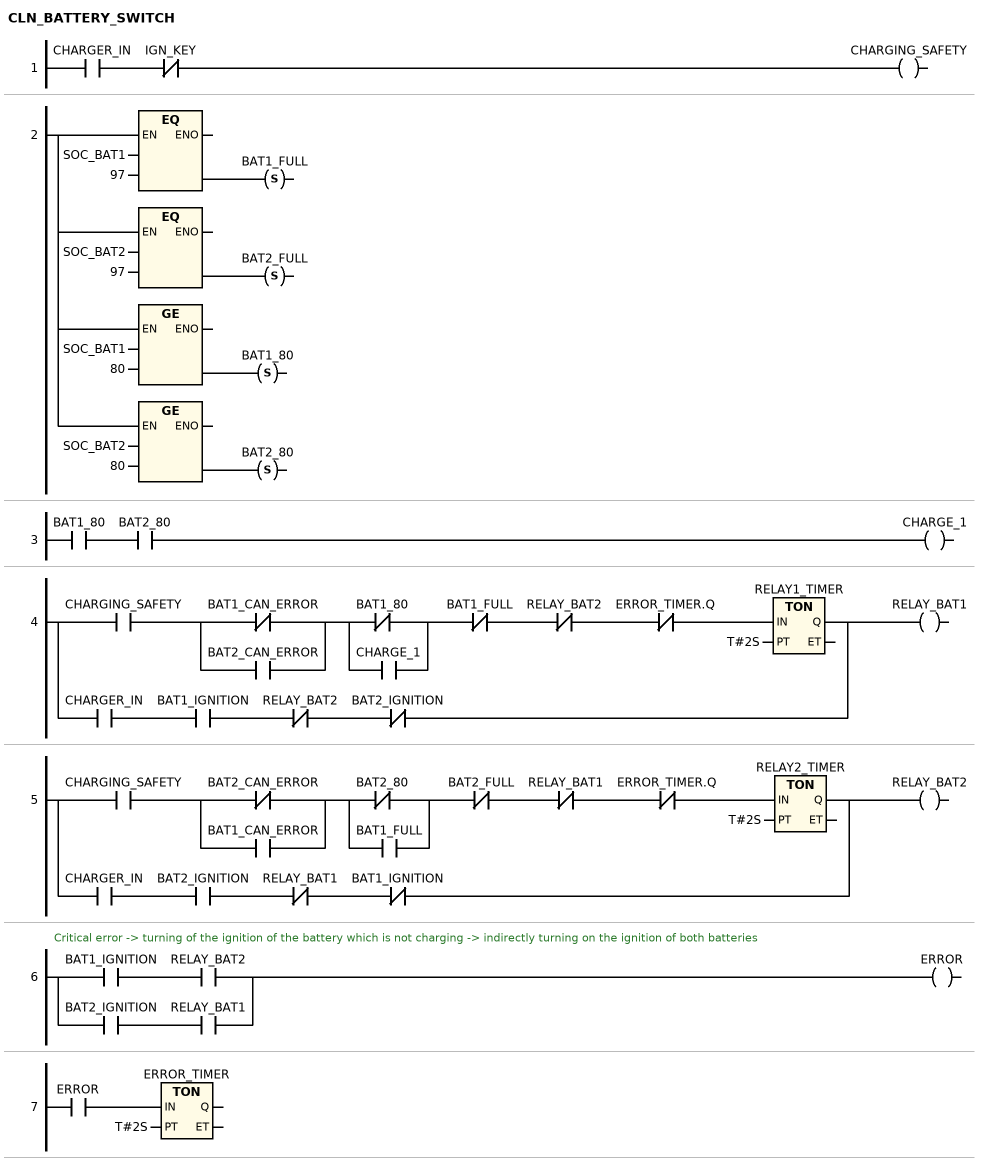
[picture p24: CLN_BATTERY_SWITCH (LD)]
_LD_ (* Ladder Diagram *)
NETWORK 1
	[CHARGER_IN] - [/IGN_KEY] --- (CHARGING_SAFETY)
NETWORK 2
	*
		EN --- EQ(SOC_BAT1, 97) => S BAT1_FULL
		EN --- EQ(SOC_BAT2, 97) => S BAT2_FULL
		EN --- GE(SOC_BAT1, 80) => S BAT1_80
		EN --- GE(SOC_BAT2, 80) => S BAT2_80
NETWORK 3
	[BAT1_80] - [BAT2_80] --- (CHARGE_1)
NETWORK 4
	{ [CHARGING_SAFETY] - { [/BAT1_CAN_ERROR] | [BAT2_CAN_ERROR] } - { [/BAT1_80] | [CHARGE_1] } - [/BAT1_FULL] - [/RELAY_BAT2] - [/ERROR_TIMER.Q] - RELAY1_TIMER:TON(IN: *, PT: T#2S) | [CHARGER_IN] - [BAT1_IGNITION] - [/RELAY_BAT2] - [/BAT2_IGNITION] } --- (RELAY_BAT1)
NETWORK 5
	{ [CHARGING_SAFETY] - { [/BAT2_CAN_ERROR] | [BAT1_CAN_ERROR] } - { [/BAT2_80] | [BAT1_FULL] } - [/BAT2_FULL] - [/RELAY_BAT1] - [/ERROR_TIMER.Q] - RELAY2_TIMER:TON(IN: *, PT: T#2S) | [CHARGER_IN] - [BAT2_IGNITION] - [/RELAY_BAT1] - [/BAT1_IGNITION] } --- (RELAY_BAT2)
NETWORK 6 (* Critical error -> turning of the ignition of the battery which is not charging -> indirectly turning on the ignition of both batteries *)
	{ [BAT1_IGNITION] - [RELAY_BAT2] | [BAT2_IGNITION] - [RELAY_BAT1] } --- (ERROR)
NETWORK 7
	[ERROR] - ERROR_TIMER:TON(IN: *, PT: T#2S)
_END_LD_
(* the same logic as Structured Text *)
(* Network 1 *)
CHARGING_SAFETY := CHARGER_IN AND NOT IGN_KEY;
(* Network 2 *)
IF SOC_BAT1 = 97 THEN BAT1_FULL := TRUE; END_IF;
IF SOC_BAT2 = 97 THEN BAT2_FULL := TRUE; END_IF;
IF SOC_BAT1 >= 80 THEN BAT1_80 := TRUE; END_IF;
IF SOC_BAT2 >= 80 THEN BAT2_80 := TRUE; END_IF;
(* Network 3 *)
CHARGE_1 := BAT1_80 AND BAT2_80;
(* Network 4 *)
RELAY1_TIMER(IN := CHARGING_SAFETY AND (NOT BAT1_CAN_ERROR OR BAT2_CAN_ERROR) AND (NOT BAT1_80 OR CHARGE_1) AND NOT BAT1_FULL AND NOT RELAY_BAT2 AND NOT ERROR_TIMER.Q, PT := T#2S);
RELAY_BAT1 := RELAY1_TIMER.Q OR CHARGER_IN AND BAT1_IGNITION AND NOT RELAY_BAT2 AND NOT BAT2_IGNITION;
(* Network 5 *)
RELAY2_TIMER(IN := CHARGING_SAFETY AND (NOT BAT2_CAN_ERROR OR BAT1_CAN_ERROR) AND (NOT BAT2_80 OR BAT1_FULL) AND NOT BAT2_FULL AND NOT RELAY_BAT1 AND NOT ERROR_TIMER.Q, PT := T#2S);
RELAY_BAT2 := RELAY2_TIMER.Q OR CHARGER_IN AND BAT2_IGNITION AND NOT RELAY_BAT1 AND NOT BAT1_IGNITION;
(* Network 6: Critical error -> turning of the ignition of the battery which is not charging -> indirectly turning on the ignition of both batteries *)
ERROR := BAT1_IGNITION AND RELAY_BAT2 OR BAT2_IGNITION AND RELAY_BAT1;
(* Network 7 *)
ERROR_TIMER(IN := ERROR, PT := T#2S);
END_FUNCTION_BLOCK

(* POU PROGRAM_FBs/CLN_CHARGING, LD *)
FUNCTION_BLOCK CLN_CHARGING
(*
THIS BLOCK IS COMPATIBLE FOR 2X CLN BATTERIES0

Created BY: Adiga
Date: 25-01-24
UPDATED :14-03-25
Version: 4
1.DUAL BATTERY CAHRGING BLOCK ONLY FOR CLN
2.UPDATED THE BLOCK FOR CHARGING WITH AND WITHOUT IGN ON
3.ADDED BATTERY CAN ERROR CODITION TO CHARGE
4.ADDED TIMER BEFORE SWITCHING BATTRY BELAY.
.
*)

VAR_INPUT
	CHANNEL: BYTE;
	CHARGER_IN: BOOL;
	IGN_KEY: BOOL;
	BAT1_IGN: BOOL;
	BAT2_IGN: BOOL;
	SOC1: BYTE;
	SOC2: BYTE;
	BAT_CAN_ERROR1: BOOL;
	BAT_CAN_ERROR2: BOOL;
	BATTERY_CHARGING: BOOL;
END_VAR

VAR_OUTPUT
	RELAY_BAT1: BOOL;
	RELAY_BAT2: BOOL;
	BLUE_LED_OUT: BOOL;
	ERROR: BOOL;
	BUZZER_ON: BOOL;
	CHARGING1: BOOL;
	CHARGING2: BOOL;
END_VAR

VAR
	CHARGE_1: BOOL;
	BAT_1_FULL: BOOL;
	BAT_2_FULL: BOOL;
	T1: TON;
	T2: TON;
	T3: TON;
	IGNITION_OFF: BOOL;
	BAT_1_80: BOOL;
	BAT_2_80: BOOL;
	FTRIG1: F_TRIG;
	TIMER5: TON;
	T4: TON;
	T5: TON;
	CHARGING_2: BLINK;
	CHARGING_1: BLINK;
END_VAR
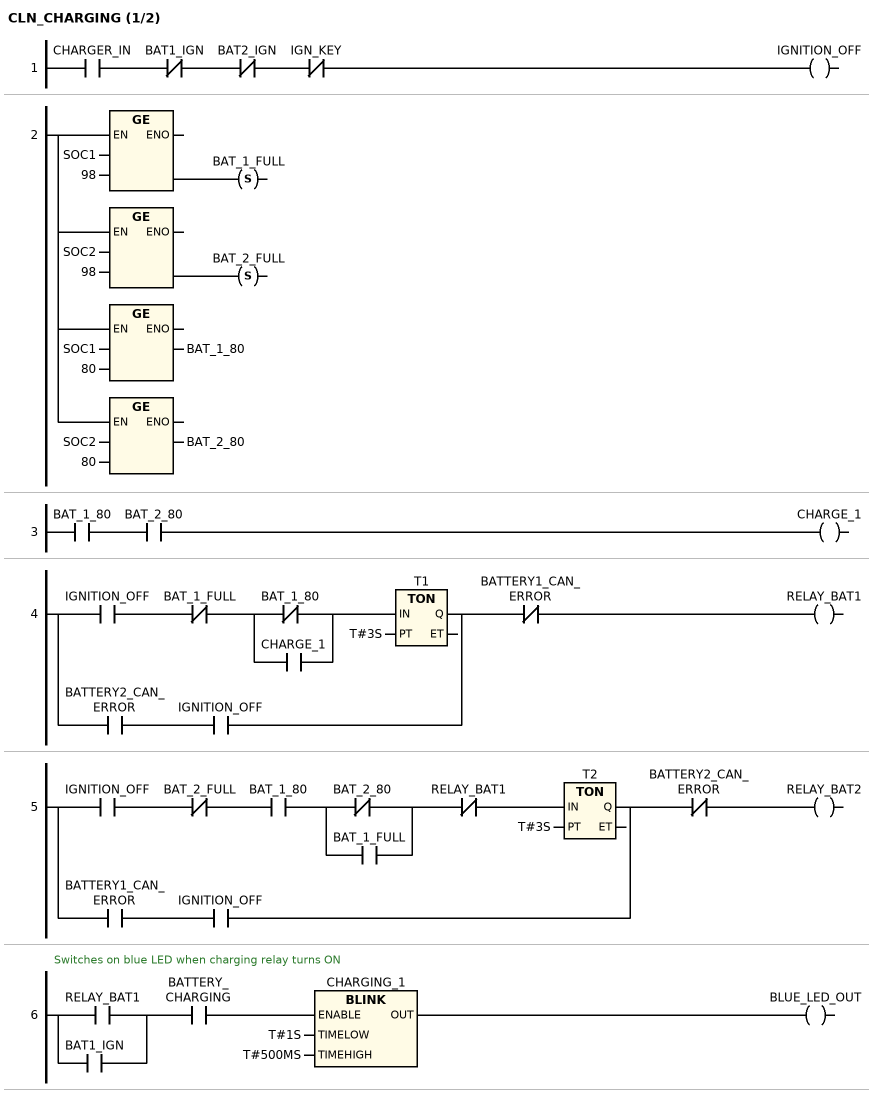
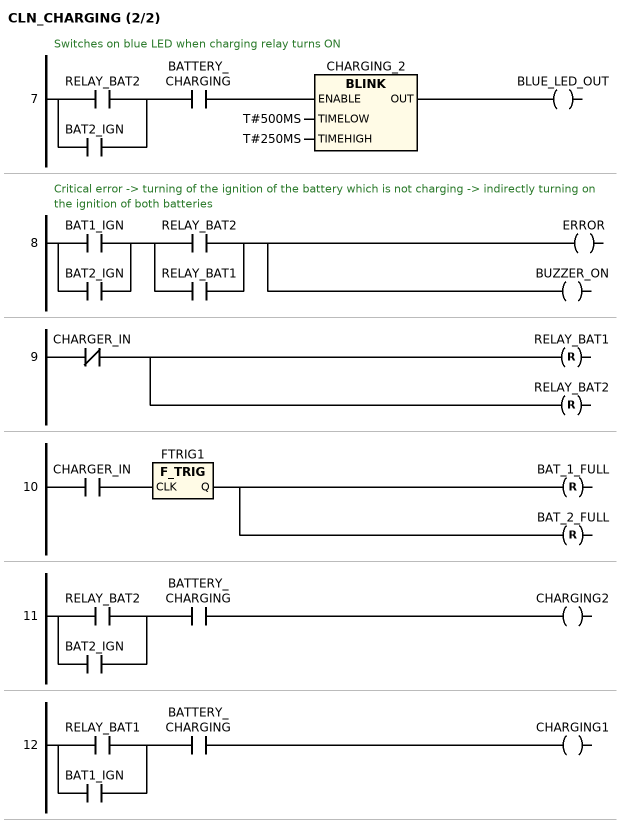
_LD_ (* Ladder Diagram *)
NETWORK 1
	[CHARGER_IN] - [/BAT1_IGN] - [/BAT2_IGN] - [/IGN_KEY] --- (IGNITION_OFF)
NETWORK 2
	*
		EN --- GE(SOC1, 98) => S BAT_1_FULL
		EN --- GE(SOC2, 98) => S BAT_2_FULL
		EN --- GE(SOC1, 80) => BAT_1_80
		EN --- GE(SOC2, 80) => BAT_2_80
NETWORK 3
	[BAT_1_80] - [BAT_2_80] --- (CHARGE_1)
NETWORK 4
	{ [IGNITION_OFF] - [/BAT_1_FULL] - { [/BAT_1_80] | [CHARGE_1] } - T1:TON(IN: *, PT: T#3S) | [BATTERY2_CAN_ERROR] - [IGNITION_OFF] } - [/BATTERY1_CAN_ERROR] --- (RELAY_BAT1)
NETWORK 5
	{ [IGNITION_OFF] - [/BAT_2_FULL] - [BAT_1_80] - { [/BAT_2_80] | [BAT_1_FULL] } - [/RELAY_BAT1] - T2:TON(IN: *, PT: T#3S) | [BATTERY1_CAN_ERROR] - [IGNITION_OFF] } - [/BATTERY2_CAN_ERROR] --- (RELAY_BAT2)
NETWORK 6 (* Switches on blue LED when charging relay turns ON *)
	{ [RELAY_BAT1] | [BAT1_IGN] } - [BATTERY_CHARGING] - CHARGING_1:BLINK(ENABLE: *, TIMELOW: T#1S, TIMEHIGH: T#500MS) --- (BLUE_LED_OUT)
NETWORK 7 (* Switches on blue LED when charging relay turns ON *)
	{ [RELAY_BAT2] | [BAT2_IGN] } - [BATTERY_CHARGING] - CHARGING_2:BLINK(ENABLE: *, TIMELOW: T#500MS, TIMEHIGH: T#250MS) --- (BLUE_LED_OUT)
NETWORK 8 (* Critical error -> turning of the ignition of the battery which is not charging -> indirectly turning on the ignition of both batteries *)
	{ [BAT1_IGN] | [BAT2_IGN] } - { [RELAY_BAT2] | [RELAY_BAT1] } --- (ERROR) (BUZZER_ON)
NETWORK 9
	[/CHARGER_IN] --- (R RELAY_BAT1) (R RELAY_BAT2)
NETWORK 10
	[CHARGER_IN] - FTRIG1:F_TRIG(CLK: *) --- (R BAT_1_FULL) (R BAT_2_FULL)
NETWORK 11
	{ [RELAY_BAT2] | [BAT2_IGN] } - [BATTERY_CHARGING] --- (CHARGING2)
NETWORK 12
	{ [RELAY_BAT1] | [BAT1_IGN] } - [BATTERY_CHARGING] --- (CHARGING1)
_END_LD_
(* the same logic as Structured Text *)
(* Network 1 *)
IGNITION_OFF := CHARGER_IN AND NOT BAT1_IGN AND NOT BAT2_IGN AND NOT IGN_KEY;
(* Network 2 *)
IF SOC1 >= 98 THEN BAT_1_FULL := TRUE; END_IF;
IF SOC2 >= 98 THEN BAT_2_FULL := TRUE; END_IF;
BAT_1_80 := SOC1 >= 80;
BAT_2_80 := SOC2 >= 80;
(* Network 3 *)
CHARGE_1 := BAT_1_80 AND BAT_2_80;
(* Network 4 *)
T1(IN := IGNITION_OFF AND NOT BAT_1_FULL AND (NOT BAT_1_80 OR CHARGE_1), PT := T#3S);
RELAY_BAT1 := (T1.Q OR BATTERY2_CAN_ERROR AND IGNITION_OFF) AND NOT BATTERY1_CAN_ERROR;
(* Network 5 *)
T2(IN := IGNITION_OFF AND NOT BAT_2_FULL AND BAT_1_80 AND (NOT BAT_2_80 OR BAT_1_FULL) AND NOT RELAY_BAT1, PT := T#3S);
RELAY_BAT2 := (T2.Q OR BATTERY1_CAN_ERROR AND IGNITION_OFF) AND NOT BATTERY2_CAN_ERROR;
(* Network 6: Switches on blue LED when charging relay turns ON *)
CHARGING_1(ENABLE := (RELAY_BAT1 OR BAT1_IGN) AND BATTERY_CHARGING, TIMELOW := T#1S, TIMEHIGH := T#500MS);
BLUE_LED_OUT := CHARGING_1.OUT;
(* Network 7: Switches on blue LED when charging relay turns ON *)
CHARGING_2(ENABLE := (RELAY_BAT2 OR BAT2_IGN) AND BATTERY_CHARGING, TIMELOW := T#500MS, TIMEHIGH := T#250MS);
BLUE_LED_OUT := CHARGING_2.OUT;
(* Network 8: Critical error -> turning of the ignition of the battery which is not charging -> indirectly turning on the ignition of both batteries *)
ERROR := (BAT1_IGN OR BAT2_IGN) AND (RELAY_BAT2 OR RELAY_BAT1);
BUZZER_ON := ERROR;
(* Network 9 *)
IF NOT CHARGER_IN THEN RELAY_BAT1 := FALSE; RELAY_BAT2 := FALSE; END_IF;
(* Network 10 *)
FTRIG1(CLK := CHARGER_IN);
IF FTRIG1.Q THEN BAT_1_FULL := FALSE; BAT_2_FULL := FALSE; END_IF;
(* Network 11 *)
CHARGING2 := (RELAY_BAT2 OR BAT2_IGN) AND BATTERY_CHARGING;
(* Network 12 *)
CHARGING1 := (RELAY_BAT1 OR BAT1_IGN) AND BATTERY_CHARGING;
END_FUNCTION_BLOCK

(* POU PROGRAM_FBs/DRIVE_LOGIC, LD *)
FUNCTION_BLOCK DRIVE_LOGIC
VAR_INPUT
	JX: INT;
	JY: INT;
	LEFT_BUTTON: BOOL;
	JOY_ORIGIN: BOOL;
	EM_SWITCH_IN: BOOL;
	OVER_TEMP: BOOL;
END_VAR
VAR_OUTPUT
	JX_1: INT;
	JY_1: INT;
	DISARM: BOOL;
	EM_BRAKE_OUT: BOOL;
	DRIVE_ERROR: BOOL;
END_VAR
VAR
	SLEEP_TIMER: TON;
	ON_DELAY: TON;
	APPLY_EM: BOOL;
	LOW_RPM: BOOL;
	EMFB_ERROR: BOOL;
END_VAR
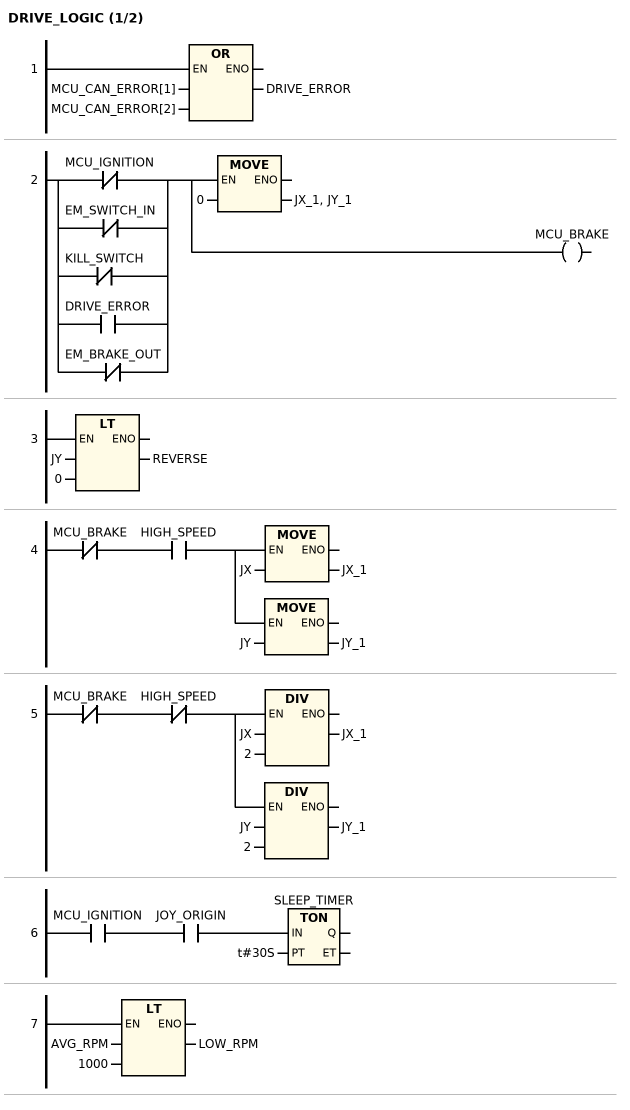
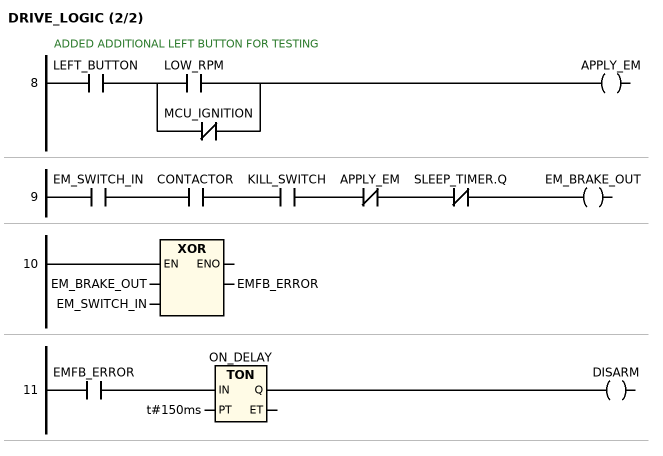
_LD_ (* Ladder Diagram *)
NETWORK 1
	*
		EN --- OR(MCU_CAN_ERROR[1], MCU_CAN_ERROR[2]) => DRIVE_ERROR
NETWORK 2
	{ [/MCU_IGNITION] | [/EM_SWITCH_IN] | [/KILL_SWITCH] | [DRIVE_ERROR] | [/EM_BRAKE_OUT] } --- (MCU_BRAKE)
		EN --- MOVE(0) => JX_1, JY_1
NETWORK 3
	*
		EN --- LT(JY, 0) => REVERSE
NETWORK 4
	[/MCU_BRAKE] - [HIGH_SPEED]
		EN --- MOVE(JX) => JX_1
		EN --- MOVE(JY) => JY_1
NETWORK 5
	[/MCU_BRAKE] - [/HIGH_SPEED]
		EN --- DIV(JX, 2) => JX_1
		EN --- DIV(JY, 2) => JY_1
NETWORK 6
	[MCU_IGNITION] - [JOY_ORIGIN] - SLEEP_TIMER:TON(IN: *, PT: t#30S)
NETWORK 7
	*
		EN --- LT(AVG_RPM, 1000) => LOW_RPM
NETWORK 8 (* ADDED ADDITIONAL LEFT BUTTON FOR TESTING *)
	[LEFT_BUTTON] - { [LOW_RPM] | [/MCU_IGNITION] } --- (APPLY_EM)
NETWORK 9
	[EM_SWITCH_IN] - [CONTACTOR] - [KILL_SWITCH] - [/APPLY_EM] - [/SLEEP_TIMER.Q] --- (EM_BRAKE_OUT)
NETWORK 10
	*
		EN --- XOR(EM_BRAKE_OUT, EM_SWITCH_IN) => EMFB_ERROR
NETWORK 11
	[EMFB_ERROR] - ON_DELAY:TON(IN: *, PT: t#150ms) --- (DISARM)
_END_LD_
(* the same logic as Structured Text *)
(* Network 1 *)
DRIVE_ERROR := MCU_CAN_ERROR[1] OR MCU_CAN_ERROR[2];
(* Network 2: see the listing above *)
(* Network 3 *)
REVERSE := JY < 0;
(* Network 4 *)
IF NOT MCU_BRAKE AND HIGH_SPEED THEN
	JX_1 := JX;
	JY_1 := JY;
END_IF;
(* Network 5 *)
IF NOT MCU_BRAKE AND NOT HIGH_SPEED THEN
	JX_1 := JX / 2;
	JY_1 := JY / 2;
END_IF;
(* Network 6 *)
SLEEP_TIMER(IN := MCU_IGNITION AND JOY_ORIGIN, PT := t#30S);
(* Network 7 *)
LOW_RPM := AVG_RPM < 1000;
(* Network 8 *)
APPLY_EM := LEFT_BUTTON AND (LOW_RPM OR NOT MCU_IGNITION);
(* Network 9 *)
EM_BRAKE_OUT := EM_SWITCH_IN AND CONTACTOR AND KILL_SWITCH AND NOT APPLY_EM AND NOT SLEEP_TIMER.Q;
(* Network 10 *)
EMFB_ERROR := EM_BRAKE_OUT XOR EM_SWITCH_IN;
(* Network 11 *)
ON_DELAY(IN := EMFB_ERROR, PT := t#150ms);
DISARM := ON_DELAY.Q;
END_FUNCTION_BLOCK

(* POU PROGRAM_FBs/DUAL_CLN_CHARGING, LD *)
FUNCTION_BLOCK DUAL_CLN_CHARGING
(*
THIS BLOCK IS COMPATIBLE FOR 2X CLN BATTERIES

Created BY: Adiga
Date: 8-08-24
Version: 1
 
*)

VAR_INPUT
	CHANNEL: BYTE;
	CHARGER_IN: BOOL;
	BAT_CAN_ERROR1: BOOL;
	BAT_CAN_ERROR2: BOOL;
	BAT1_IGN: BOOL;
	BAT2_IGN: BOOL;
	BATTERY_CHARGING: BOOL;

END_VAR

VAR_OUTPUT
	RELAY_BAT1: BOOL;
	RELAY_BAT2: BOOL;
	BLUE_LED_OUT: BOOL;
	ERROR: BOOL;
	BUZZER_ON: BOOL;
	CHARGING1: BOOL;
	CHARGING2: BOOL;
END_VAR

VAR
	CHARGE_1: BOOL;
	BAT_1_FULL: BOOL;
	BAT_2_FULL: BOOL;
	RX_SOLTERRA: RX_CAN;
	CHARGER_TIMER: TON;
	SOLTERRA_TX: CAN_TX;
	CHARGING_FRAME: ARRAY [0..7] OF BYTE  := 16#03,16#25,16#01,16#5E,0,0,0,0;

	T1: TON;
	T2: TON;
	T3: TON;
	SOC2: BYTE;
	SOC1: BYTE;
	TX_CLN: CAN_TX;
	IGNITION_OFF: BOOL;
	BAT_1_80: BOOL;
	BAT_2_80: BOOL;
	FTRIG1: F_TRIG;
	TIMER5: TON;
	T4: TON;
	T5: TON;

	CHARGE: F_TRIG;
END_VAR
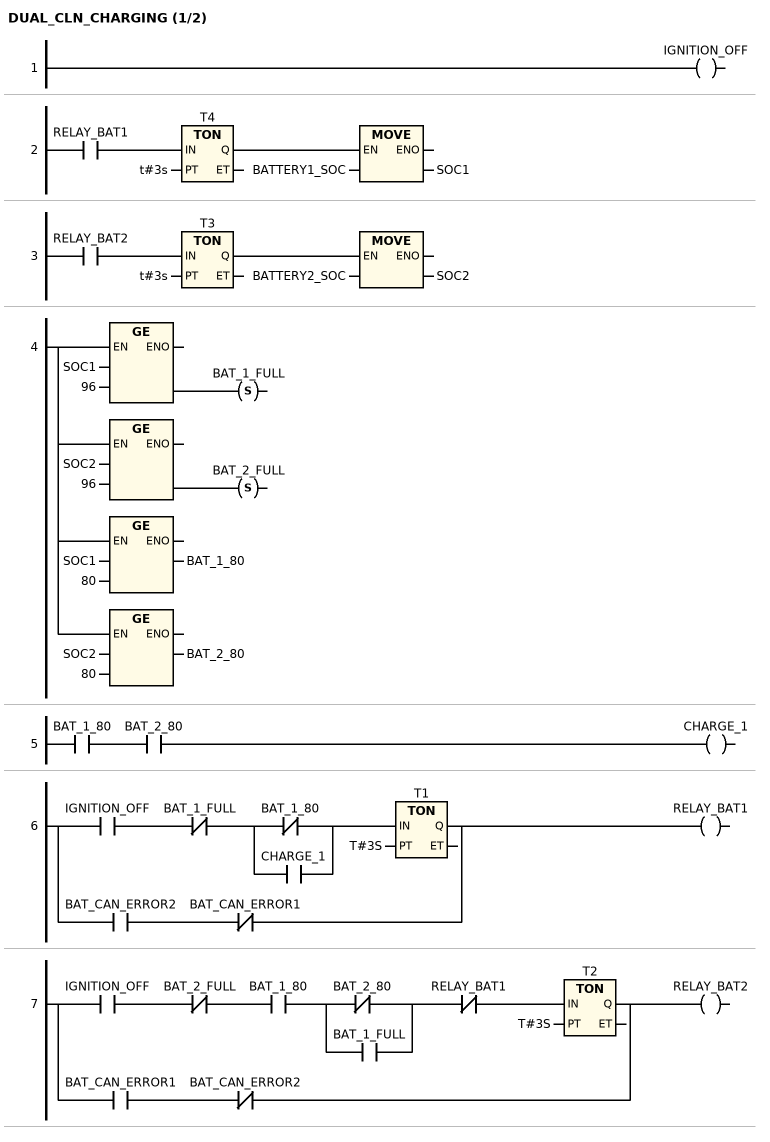
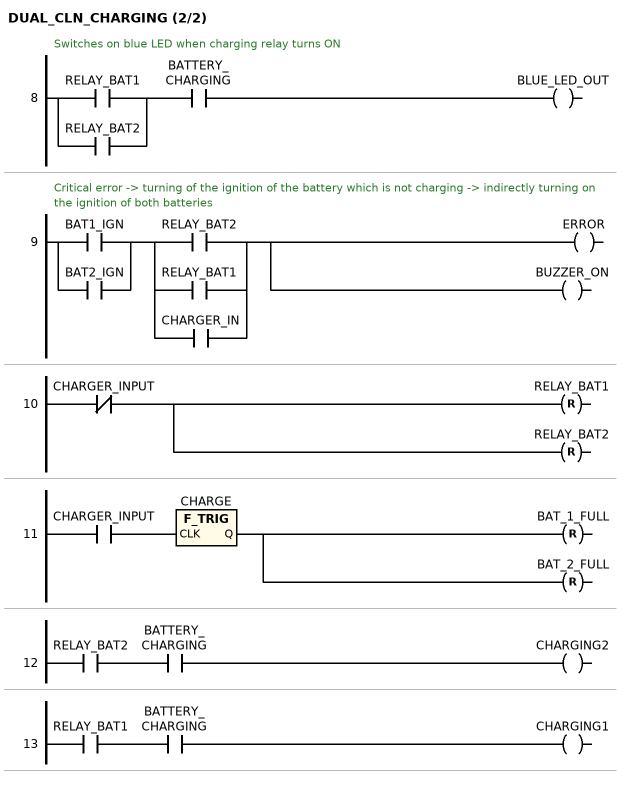
_LD_ (* Ladder Diagram *)
NETWORK 1
	* --- (IGNITION_OFF)
NETWORK 2
	[RELAY_BAT1] - T4:TON(IN: *, PT: t#3s)
		EN --- MOVE(BATTERY1_SOC) => SOC1
NETWORK 3
	[RELAY_BAT2] - T3:TON(IN: *, PT: t#3s)
		EN --- MOVE(BATTERY2_SOC) => SOC2
NETWORK 4
	*
		EN --- GE(SOC1, 96) => S BAT_1_FULL
		EN --- GE(SOC2, 96) => S BAT_2_FULL
		EN --- GE(SOC1, 80) => BAT_1_80
		EN --- GE(SOC2, 80) => BAT_2_80
NETWORK 5
	[BAT_1_80] - [BAT_2_80] --- (CHARGE_1)
NETWORK 6
	{ [IGNITION_OFF] - [/BAT_1_FULL] - { [/BAT_1_80] | [CHARGE_1] } - T1:TON(IN: *, PT: T#3S) | [BAT_CAN_ERROR2] - [/BAT_CAN_ERROR1] } --- (RELAY_BAT1)
NETWORK 7
	{ [IGNITION_OFF] - [/BAT_2_FULL] - [BAT_1_80] - { [/BAT_2_80] | [BAT_1_FULL] } - [/RELAY_BAT1] - T2:TON(IN: *, PT: T#3S) | [BAT_CAN_ERROR1] - [/BAT_CAN_ERROR2] } --- (RELAY_BAT2)
NETWORK 8 (* Switches on blue LED when charging relay turns ON *)
	{ [RELAY_BAT1] | [RELAY_BAT2] } - [BATTERY_CHARGING] --- (BLUE_LED_OUT)
NETWORK 9 (* Critical error -> turning of the ignition of the battery which is not charging -> indirectly turning on the ignition of both batteries *)
	{ [BAT1_IGN] | [BAT2_IGN] } - { [RELAY_BAT2] | [RELAY_BAT1] | [CHARGER_IN] } --- (ERROR) (BUZZER_ON)
NETWORK 10
	[/CHARGER_INPUT] --- (R RELAY_BAT1) (R RELAY_BAT2)
NETWORK 11
	[CHARGER_INPUT] - CHARGE:F_TRIG(CLK: *) --- (R BAT_1_FULL) (R BAT_2_FULL)
NETWORK 12
	[RELAY_BAT2] - [BATTERY_CHARGING] --- (CHARGING2)
NETWORK 13
	[RELAY_BAT1] - [BATTERY_CHARGING] --- (CHARGING1)
_END_LD_
(* the same logic as Structured Text *)
(* Network 1 *)
IGNITION_OFF := TRUE;
(* Network 2 *)
T4(IN := RELAY_BAT1, PT := t#3s);
IF T4.Q THEN
	SOC1 := BATTERY1_SOC;
END_IF;
(* Network 3 *)
T3(IN := RELAY_BAT2, PT := t#3s);
IF T3.Q THEN
	SOC2 := BATTERY2_SOC;
END_IF;
(* Network 4 *)
IF SOC1 >= 96 THEN BAT_1_FULL := TRUE; END_IF;
IF SOC2 >= 96 THEN BAT_2_FULL := TRUE; END_IF;
BAT_1_80 := SOC1 >= 80;
BAT_2_80 := SOC2 >= 80;
(* Network 5 *)
CHARGE_1 := BAT_1_80 AND BAT_2_80;
(* Network 6 *)
T1(IN := IGNITION_OFF AND NOT BAT_1_FULL AND (NOT BAT_1_80 OR CHARGE_1), PT := T#3S);
RELAY_BAT1 := T1.Q OR BAT_CAN_ERROR2 AND NOT BAT_CAN_ERROR1;
(* Network 7 *)
T2(IN := IGNITION_OFF AND NOT BAT_2_FULL AND BAT_1_80 AND (NOT BAT_2_80 OR BAT_1_FULL) AND NOT RELAY_BAT1, PT := T#3S);
RELAY_BAT2 := T2.Q OR BAT_CAN_ERROR1 AND NOT BAT_CAN_ERROR2;
(* Network 8: Switches on blue LED when charging relay turns ON *)
BLUE_LED_OUT := (RELAY_BAT1 OR RELAY_BAT2) AND BATTERY_CHARGING;
(* Network 9: Critical error -> turning of the ignition of the battery which is not charging -> indirectly turning on the ignition of both batteries *)
ERROR := (BAT1_IGN OR BAT2_IGN) AND (RELAY_BAT2 OR RELAY_BAT1 OR CHARGER_IN);
BUZZER_ON := ERROR;
(* Network 10 *)
IF NOT CHARGER_INPUT THEN RELAY_BAT1 := FALSE; RELAY_BAT2 := FALSE; END_IF;
(* Network 11 *)
CHARGE(CLK := CHARGER_INPUT);
IF CHARGE.Q THEN BAT_1_FULL := FALSE; BAT_2_FULL := FALSE; END_IF;
(* Network 12 *)
CHARGING2 := RELAY_BAT2 AND BATTERY_CHARGING;
(* Network 13 *)
CHARGING1 := RELAY_BAT1 AND BATTERY_CHARGING;
END_FUNCTION_BLOCK

(* POU FB_LIBRARY/DWORD_BYTE_CONVERSION, FBD *)
FUNCTION_BLOCK DWORD_BYTE_CONVERSION
(* BYTE_0 : LSB    ---------   BYTE_3 : MSB *)
VAR_INPUT
	INPUT_DWORD: DWORD;
END_VAR
VAR_OUTPUT
	BYTE_0: BYTE;
	BYTE_1: BYTE;
	BYTE_2: BYTE;
	BYTE_3: BYTE;
END_VAR
VAR
	WORD_1: WORD;
	WORD_2: WORD;
END_VAR
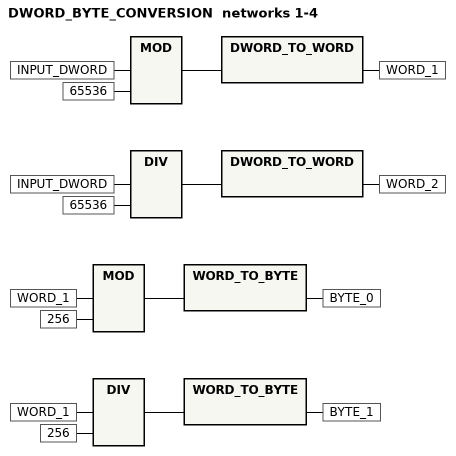
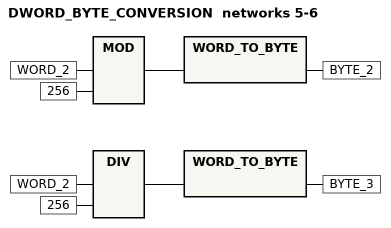
_FBD_ (* Function Block Diagram *)
NETWORK 1
	DWORD_TO_WORD(MOD(INPUT_DWORD, 65536)) => WORD_1
NETWORK 2
	DWORD_TO_WORD(DIV(INPUT_DWORD, 65536)) => WORD_2
NETWORK 3
	WORD_TO_BYTE(MOD(WORD_1, 256)) => BYTE_0
NETWORK 4
	WORD_TO_BYTE(DIV(WORD_1, 256)) => BYTE_1
NETWORK 5
	WORD_TO_BYTE(MOD(WORD_2, 256)) => BYTE_2
NETWORK 6
	WORD_TO_BYTE(DIV(WORD_2, 256)) => BYTE_3
_END_FBD_
(* the same logic as Structured Text *)
(* Network 1 *)
WORD_1 := DWORD_TO_WORD(INPUT_DWORD MOD 65536);
(* Network 2 *)
WORD_2 := DWORD_TO_WORD(INPUT_DWORD / 65536);
(* Network 3 *)
BYTE_0 := WORD_TO_BYTE(WORD_1 MOD 256);
(* Network 4 *)
BYTE_1 := WORD_TO_BYTE(WORD_1 / 256);
(* Network 5 *)
BYTE_2 := WORD_TO_BYTE(WORD_2 MOD 256);
(* Network 6 *)
BYTE_3 := WORD_TO_BYTE(WORD_2 / 256);
END_FUNCTION_BLOCK

(* POU PROGRAM_FBs/HYDRAULIC_CONTROL, LD *)
FUNCTION_BLOCK HYDRAULIC_CONTROL
VAR_INPUT
	DEADMAN: BOOL;
END_VAR
VAR_OUTPUT
END_VAR
VAR
	HYD_SPEED: INT;
	IDLE_MODE: BOOL;
	CUTOFF: INT;
	STATISTICS: STATISTICS_INT;
	RESET_AVG: BOOL;
	T1: TON;
	TRIG_1: R_TRIG;
	T2: TON;
	RUNNING_AVG: INT:=0;
	SET_IDLE: BOOL;
	HIGH_RPM: BOOL;
	WAIT: BOOL;
	UPPER_LIMIT: INT;
	MCU_RX_6: CHARA_MCU_RX;
	MCU_TX_6: CHARA_MCU_TX;
END_VAR
VAR CONSTANT
	IDLE_SPEED: INT :=0;
	ECO_CUTOFF: INT := 70;
	POWER_CUTOFF: INT := 90;
	BUFFER: INT := 10;
	HYD_RAMP: INT:= 100;
	MCU_RAMP: BYTE := 5;
	PHASE_LIMIT: BYTE := 60;
END_VAR
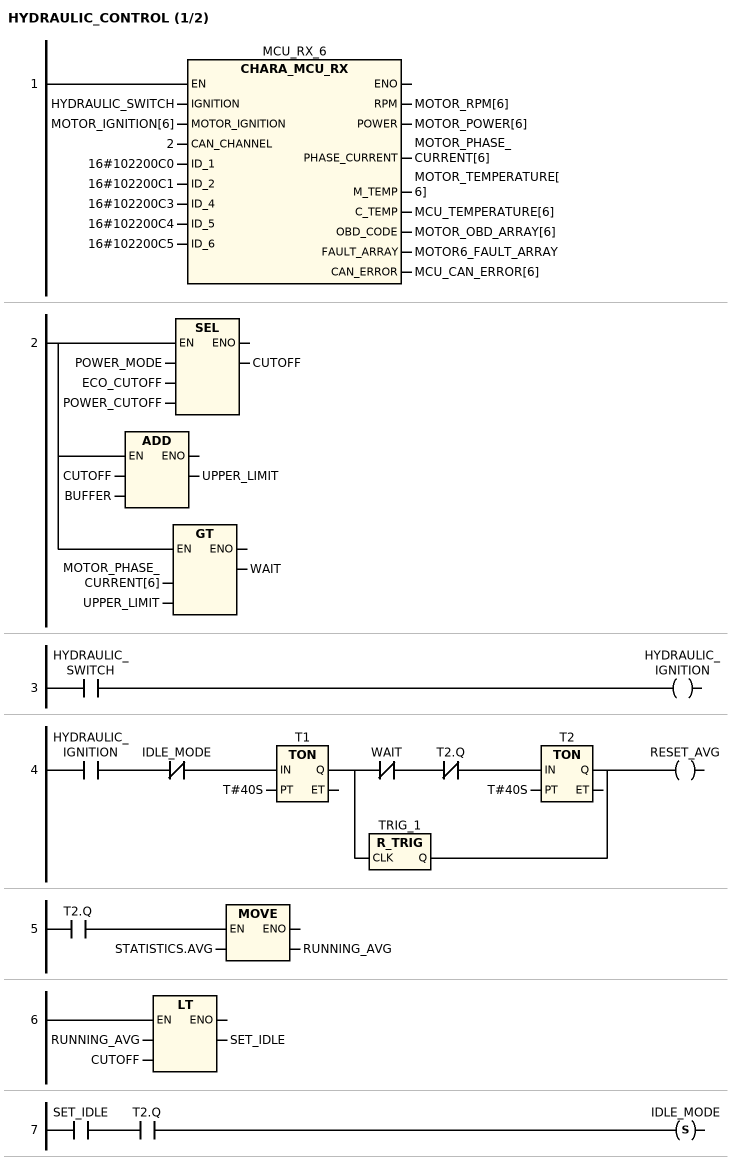
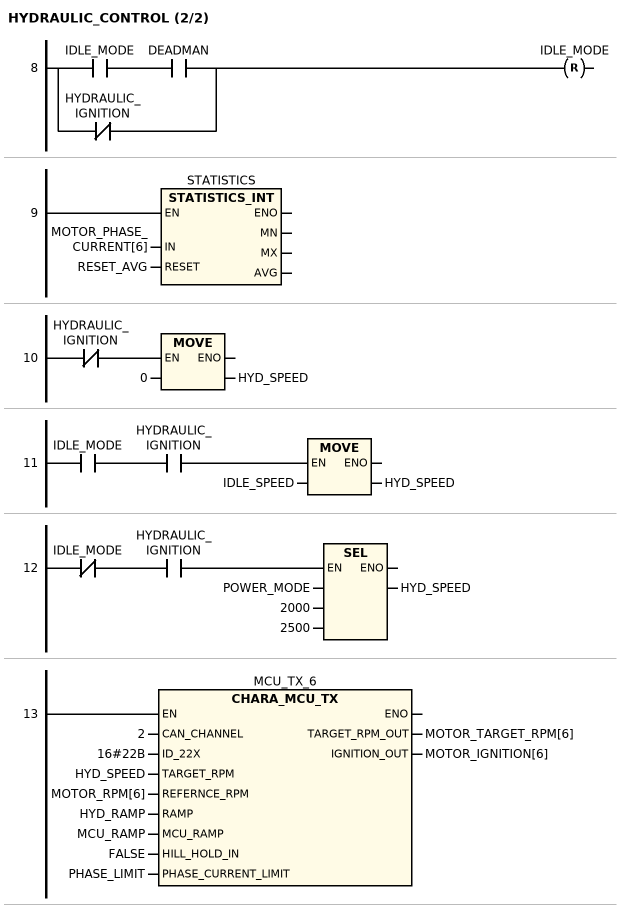
_LD_ (* Ladder Diagram *)
NETWORK 1
	*
		EN --- MCU_RX_6:CHARA_MCU_RX(IGNITION: HYDRAULIC_SWITCH, MOTOR_IGNITION: MOTOR_IGNITION[6], CAN_CHANNEL: 2, ID_1: 16#102200C0, ID_2: 16#102200C1, ID_4: 16#102200C3, ID_5: 16#102200C4, ID_6: 16#102200C5, POWER => MOTOR_POWER[6], PHASE_CURRENT => MOTOR_PHASE_CURRENT[6], M_TEMP => MOTOR_TEMPERATURE[6], C_TEMP => MCU_TEMPERATURE[6], OBD_CODE => MOTOR_OBD_ARRAY[6], FAULT_ARRAY => MOTOR6_FAULT_ARRAY, CAN_ERROR => MCU_CAN_ERROR[6]) => MOTOR_RPM[6]
NETWORK 2
	*
		EN --- SEL(POWER_MODE, ECO_CUTOFF, POWER_CUTOFF) => CUTOFF
		EN --- ADD(CUTOFF, BUFFER) => UPPER_LIMIT
		EN --- GT(MOTOR_PHASE_CURRENT[6], UPPER_LIMIT) => WAIT
NETWORK 3
	[HYDRAULIC_SWITCH] --- (HYDRAULIC_IGNITION)
NETWORK 4
	[HYDRAULIC_IGNITION] - [/IDLE_MODE] - T1:TON(IN: *, PT: T#40S) - { [/WAIT] - [/T2.Q] - T2:TON(IN: *, PT: T#40S) | TRIG_1:R_TRIG(CLK: *) } --- (RESET_AVG)
NETWORK 5
	[T2.Q]
		EN --- MOVE(STATISTICS.AVG) => RUNNING_AVG
NETWORK 6
	*
		EN --- LT(RUNNING_AVG, CUTOFF) => SET_IDLE
NETWORK 7
	[SET_IDLE] - [T2.Q] --- (S IDLE_MODE)
NETWORK 8
	{ [IDLE_MODE] - [DEADMAN] | [/HYDRAULIC_IGNITION] } --- (R IDLE_MODE)
NETWORK 9
	*
		EN --- STATISTICS:STATISTICS_INT(IN: MOTOR_PHASE_CURRENT[6], RESET: RESET_AVG)
NETWORK 10
	[/HYDRAULIC_IGNITION]
		EN --- MOVE(0) => HYD_SPEED
NETWORK 11
	[IDLE_MODE] - [HYDRAULIC_IGNITION]
		EN --- MOVE(IDLE_SPEED) => HYD_SPEED
NETWORK 12
	[/IDLE_MODE] - [HYDRAULIC_IGNITION]
		EN --- SEL(POWER_MODE, 2000, 2500) => HYD_SPEED
NETWORK 13
	*
		EN --- MCU_TX_6:CHARA_MCU_TX(CAN_CHANNEL: 2, ID_22X: 16#22B, TARGET_RPM: HYD_SPEED, REFERNCE_RPM: MOTOR_RPM[6], RAMP: HYD_RAMP, MCU_RAMP: MCU_RAMP, HILL_HOLD_IN: FALSE, PHASE_CURRENT_LIMIT: PHASE_LIMIT, IGNITION_OUT => MOTOR_IGNITION[6]) => MOTOR_TARGET_RPM[6]
_END_LD_
(* the same logic as Structured Text *)
(* Network 1 *)
MCU_RX_6(IGNITION := HYDRAULIC_SWITCH, MOTOR_IGNITION := MOTOR_IGNITION[6], CAN_CHANNEL := 2, ID_1 := 16#102200C0, ID_2 := 16#102200C1, ID_4 := 16#102200C3, ID_5 := 16#102200C4, ID_6 := 16#102200C5);
MOTOR_POWER[6] := MCU_RX_6.POWER;
MOTOR_PHASE_CURRENT[6] := MCU_RX_6.PHASE_CURRENT;
MOTOR_TEMPERATURE[6] := MCU_RX_6.M_TEMP;
MCU_TEMPERATURE[6] := MCU_RX_6.C_TEMP;
MOTOR_OBD_ARRAY[6] := MCU_RX_6.OBD_CODE;
MOTOR6_FAULT_ARRAY := MCU_RX_6.FAULT_ARRAY;
MCU_CAN_ERROR[6] := MCU_RX_6.CAN_ERROR;
MOTOR_RPM[6] := MCU_RX_6.RPM;
(* Network 2 *)
CUTOFF := SEL(POWER_MODE, ECO_CUTOFF, POWER_CUTOFF);
UPPER_LIMIT := CUTOFF + BUFFER;
WAIT := MOTOR_PHASE_CURRENT[6] > UPPER_LIMIT;
(* Network 3 *)
HYDRAULIC_IGNITION := HYDRAULIC_SWITCH;
(* Network 4 *)
T1(IN := HYDRAULIC_IGNITION AND NOT IDLE_MODE, PT := T#40S);
T2(IN := T1.Q AND NOT WAIT AND NOT T2.Q, PT := T#40S);
TRIG_1(CLK := T1.Q);
RESET_AVG := T2.Q OR TRIG_1.Q;
(* Network 5 *)
IF T2.Q THEN
	RUNNING_AVG := STATISTICS.AVG;
END_IF;
(* Network 6 *)
SET_IDLE := RUNNING_AVG < CUTOFF;
(* Network 7 *)
IF SET_IDLE AND T2.Q THEN IDLE_MODE := TRUE; END_IF;
(* Network 8 *)
IF IDLE_MODE AND DEADMAN OR NOT HYDRAULIC_IGNITION THEN IDLE_MODE := FALSE; END_IF;
(* Network 9 *)
STATISTICS(IN := MOTOR_PHASE_CURRENT[6], RESET := RESET_AVG);
(* Network 10 *)
IF NOT HYDRAULIC_IGNITION THEN
	HYD_SPEED := 0;
END_IF;
(* Network 11 *)
IF IDLE_MODE AND HYDRAULIC_IGNITION THEN
	HYD_SPEED := IDLE_SPEED;
END_IF;
(* Network 12 *)
IF NOT IDLE_MODE AND HYDRAULIC_IGNITION THEN
	HYD_SPEED := SEL(POWER_MODE, 2000, 2500);
END_IF;
(* Network 13 *)
MCU_TX_6(CAN_CHANNEL := 2, ID_22X := 16#22B, TARGET_RPM := HYD_SPEED, REFERNCE_RPM := MOTOR_RPM[6], RAMP := HYD_RAMP, MCU_RAMP := MCU_RAMP, HILL_HOLD_IN := FALSE, PHASE_CURRENT_LIMIT := PHASE_LIMIT);
MOTOR_IGNITION[6] := MCU_TX_6.IGNITION_OUT;
MOTOR_TARGET_RPM[6] := MCU_TX_6.TARGET_RPM_OUT;
END_FUNCTION_BLOCK

(* POU PROGRAM_FBs/IMU_SENSOR, LD *)
FUNCTION_BLOCK IMU_SENSOR

(*
	Created BY: Adiga
Date: 2-07-24
Version: 1
Updated BY: ADIGA
1.

*)
VAR_INPUT
END_VAR
VAR_OUTPUT
	IMY_X_OUT: BYTE;
	IMU_Y_OUT: BYTE;
	ALERT: BOOL;
END_VAR
VAR
	RX_18C: RX_CAN;
	X_ANGLE_WORD: WORD;
	X_ANGLE: INT;

	Y_ANGLE_WORD: WORD;
	Y_ANGLE: INT;

	Y_IMU: INT;
	X_IMU: INT;

	TON_IMU: TON;
	Y_ALERT: BOOL;
	PAST_TIMER: TON;
	Y_PAST: INT;
	STORE_Y_MAX: BOOL;
	X_PAST: INT;
	STORE_X_MAX: BOOL;
	STORE_Y_MIN: BOOL;
	STORE_X_MIN: BOOL;
	X_ALERT: BOOL;
	BUZZER_SOUND: BLINK;
	IMU_BUZZER: BOOL;
END_VAR
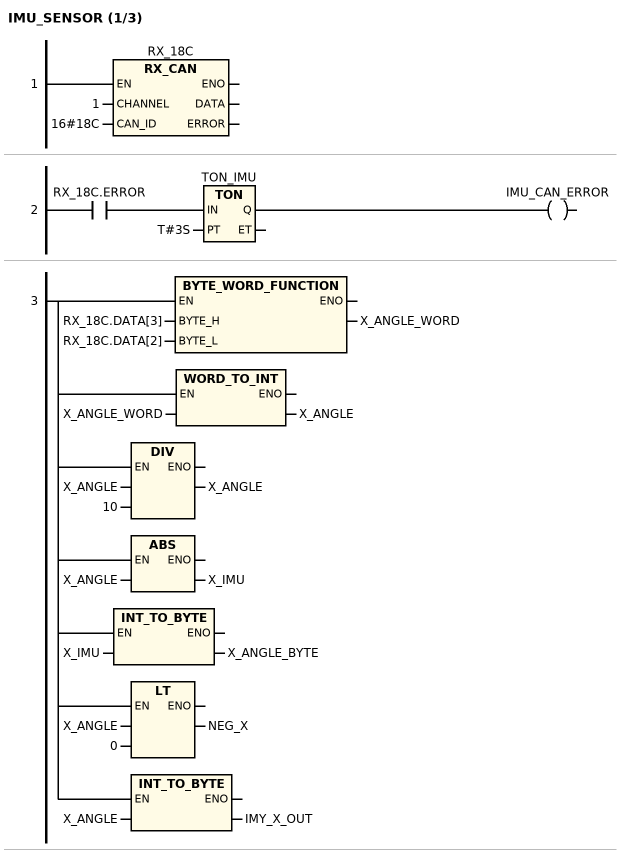
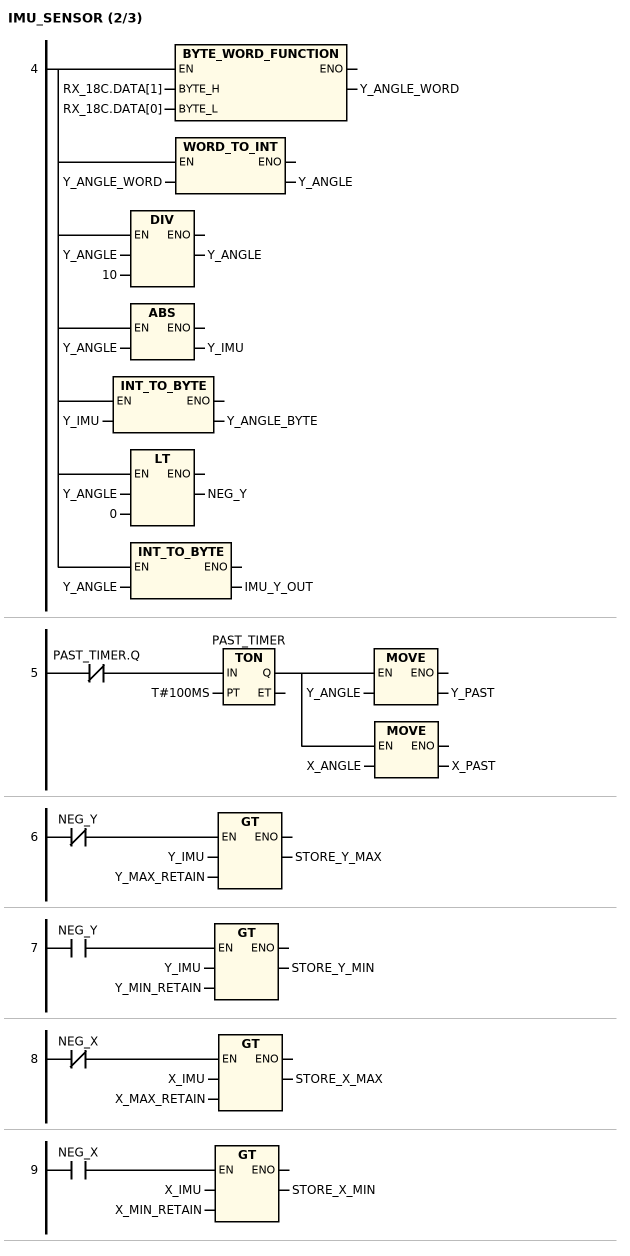
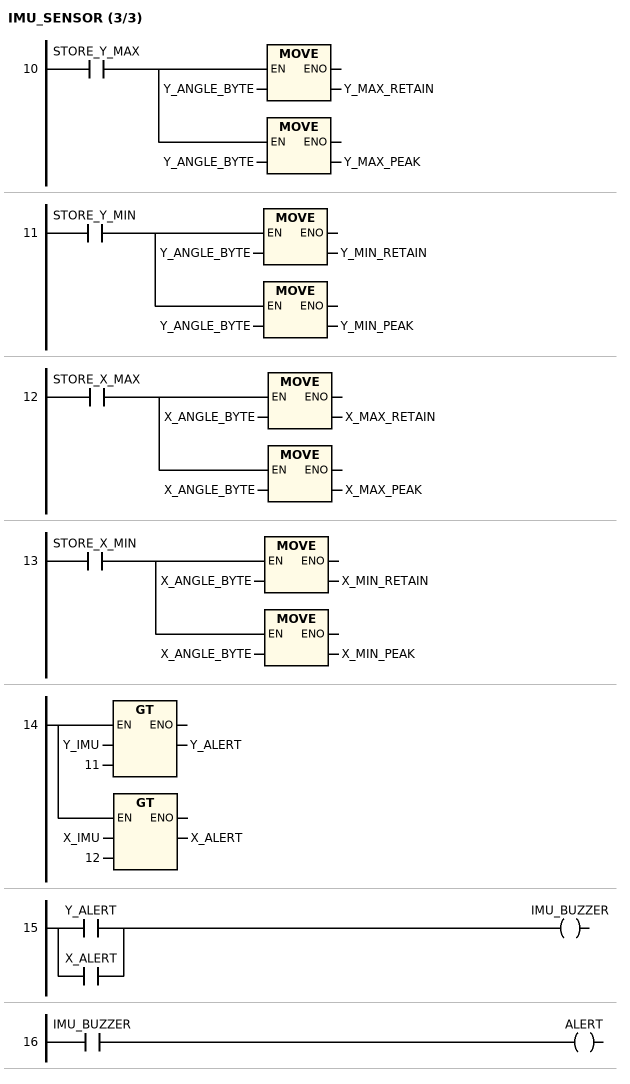
_LD_ (* Ladder Diagram *)
NETWORK 1
	*
		EN --- RX_18C:RX_CAN(CHANNEL: 1, CAN_ID: 16#18C)
NETWORK 2
	[RX_18C.ERROR] - TON_IMU:TON(IN: *, PT: T#3S) --- (IMU_CAN_ERROR)
NETWORK 3
	*
		EN --- BYTE_WORD_FUNCTION(BYTE_H: RX_18C.DATA[3], BYTE_L: RX_18C.DATA[2]) => X_ANGLE_WORD
		EN --- WORD_TO_INT(X_ANGLE_WORD) => X_ANGLE
		EN --- DIV(X_ANGLE, 10) => X_ANGLE
		EN --- ABS(X_ANGLE) => X_IMU
		EN --- INT_TO_BYTE(X_IMU) => X_ANGLE_BYTE
		EN --- LT(X_ANGLE, 0) => NEG_X
		EN --- INT_TO_BYTE(X_ANGLE) => IMY_X_OUT
NETWORK 4
	*
		EN --- BYTE_WORD_FUNCTION(BYTE_H: RX_18C.DATA[1], BYTE_L: RX_18C.DATA[0]) => Y_ANGLE_WORD
		EN --- WORD_TO_INT(Y_ANGLE_WORD) => Y_ANGLE
		EN --- DIV(Y_ANGLE, 10) => Y_ANGLE
		EN --- ABS(Y_ANGLE) => Y_IMU
		EN --- INT_TO_BYTE(Y_IMU) => Y_ANGLE_BYTE
		EN --- LT(Y_ANGLE, 0) => NEG_Y
		EN --- INT_TO_BYTE(Y_ANGLE) => IMU_Y_OUT
NETWORK 5
	[/PAST_TIMER.Q] - PAST_TIMER:TON(IN: *, PT: T#100MS)
		EN --- MOVE(Y_ANGLE) => Y_PAST
		EN --- MOVE(X_ANGLE) => X_PAST
NETWORK 6
	[/NEG_Y]
		EN --- GT(Y_IMU, Y_MAX_RETAIN) => STORE_Y_MAX
NETWORK 7
	[NEG_Y]
		EN --- GT(Y_IMU, Y_MIN_RETAIN) => STORE_Y_MIN
NETWORK 8
	[/NEG_X]
		EN --- GT(X_IMU, X_MAX_RETAIN) => STORE_X_MAX
NETWORK 9
	[NEG_X]
		EN --- GT(X_IMU, X_MIN_RETAIN) => STORE_X_MIN
NETWORK 10
	[STORE_Y_MAX]
		EN --- MOVE(Y_ANGLE_BYTE) => Y_MAX_RETAIN
		EN --- MOVE(Y_ANGLE_BYTE) => Y_MAX_PEAK
NETWORK 11
	[STORE_Y_MIN]
		EN --- MOVE(Y_ANGLE_BYTE) => Y_MIN_RETAIN
		EN --- MOVE(Y_ANGLE_BYTE) => Y_MIN_PEAK
NETWORK 12
	[STORE_X_MAX]
		EN --- MOVE(X_ANGLE_BYTE) => X_MAX_RETAIN
		EN --- MOVE(X_ANGLE_BYTE) => X_MAX_PEAK
NETWORK 13
	[STORE_X_MIN]
		EN --- MOVE(X_ANGLE_BYTE) => X_MIN_RETAIN
		EN --- MOVE(X_ANGLE_BYTE) => X_MIN_PEAK
NETWORK 14
	*
		EN --- GT(Y_IMU, 11) => Y_ALERT
		EN --- GT(X_IMU, 12) => X_ALERT
NETWORK 15
	{ [Y_ALERT] | [X_ALERT] } --- (IMU_BUZZER)
NETWORK 16
	[IMU_BUZZER] --- (ALERT)
_END_LD_
(* the same logic as Structured Text *)
(* Network 1 *)
RX_18C(CHANNEL := 1, CAN_ID := 16#18C);
(* Network 2 *)
TON_IMU(IN := RX_18C.ERROR, PT := T#3S);
IMU_CAN_ERROR := TON_IMU.Q;
(* Network 3 *)
X_ANGLE_WORD := BYTE_WORD_FUNCTION(BYTE_H := RX_18C.DATA[3], BYTE_L := RX_18C.DATA[2]);
X_ANGLE := WORD_TO_INT(X_ANGLE_WORD);
X_ANGLE := X_ANGLE / 10;
X_IMU := ABS(X_ANGLE);
X_ANGLE_BYTE := INT_TO_BYTE(X_IMU);
NEG_X := X_ANGLE < 0;
IMY_X_OUT := INT_TO_BYTE(X_ANGLE);
(* Network 4 *)
Y_ANGLE_WORD := BYTE_WORD_FUNCTION(BYTE_H := RX_18C.DATA[1], BYTE_L := RX_18C.DATA[0]);
Y_ANGLE := WORD_TO_INT(Y_ANGLE_WORD);
Y_ANGLE := Y_ANGLE / 10;
Y_IMU := ABS(Y_ANGLE);
Y_ANGLE_BYTE := INT_TO_BYTE(Y_IMU);
NEG_Y := Y_ANGLE < 0;
IMU_Y_OUT := INT_TO_BYTE(Y_ANGLE);
(* Network 5 *)
PAST_TIMER(IN := NOT PAST_TIMER.Q, PT := T#100MS);
IF PAST_TIMER.Q THEN
	Y_PAST := Y_ANGLE;
	X_PAST := X_ANGLE;
END_IF;
(* Network 6 *)
IF NOT NEG_Y THEN
	STORE_Y_MAX := Y_IMU > Y_MAX_RETAIN;
END_IF;
(* Network 7 *)
IF NEG_Y THEN
	STORE_Y_MIN := Y_IMU > Y_MIN_RETAIN;
END_IF;
(* Network 8 *)
IF NOT NEG_X THEN
	STORE_X_MAX := X_IMU > X_MAX_RETAIN;
END_IF;
(* Network 9 *)
IF NEG_X THEN
	STORE_X_MIN := X_IMU > X_MIN_RETAIN;
END_IF;
(* Network 10 *)
IF STORE_Y_MAX THEN
	Y_MAX_RETAIN := Y_ANGLE_BYTE;
	Y_MAX_PEAK := Y_ANGLE_BYTE;
END_IF;
(* Network 11 *)
IF STORE_Y_MIN THEN
	Y_MIN_RETAIN := Y_ANGLE_BYTE;
	Y_MIN_PEAK := Y_ANGLE_BYTE;
END_IF;
(* Network 12 *)
IF STORE_X_MAX THEN
	X_MAX_RETAIN := X_ANGLE_BYTE;
	X_MAX_PEAK := X_ANGLE_BYTE;
END_IF;
(* Network 13 *)
IF STORE_X_MIN THEN
	X_MIN_RETAIN := X_ANGLE_BYTE;
	X_MIN_PEAK := X_ANGLE_BYTE;
END_IF;
(* Network 14 *)
Y_ALERT := Y_IMU > 11;
X_ALERT := X_IMU > 12;
(* Network 15 *)
IMU_BUZZER := Y_ALERT OR X_ALERT;
(* Network 16 *)
ALERT := IMU_BUZZER;
END_FUNCTION_BLOCK

(* POU EXCLUDES/IMU_SENSOR_HOLD, LD *)
FUNCTION_BLOCK IMU_SENSOR_HOLD
VAR_OUTPUT
	IMY_X_OUT: BYTE;
	IMU_Y_OUT: BYTE;
	IMU_BUZZER_ALERT: BOOL;
END_VAR
VAR
	RX_18C: RX_CAN;
	X_ANGLE_WORD: WORD;
	X_ANGLE: INT;
	Y_ANGLE_WORD: WORD;
	Y_ANGLE: INT;
	Y_IMU: INT;
	X_IMU: INT;
	TON_IMU: TON;
	Y_ALERT: BOOL;
	X_ALERT: BOOL;
	PAST_TIMER: TON;
	Y_PAST: INT;
	STORE_Y_MAX: BOOL;
	X_PAST: INT;
	STORE_X_MAX: BOOL;
	STORE_Y_MIN: BOOL;
	STORE_X_MIN: BOOL;
END_VAR
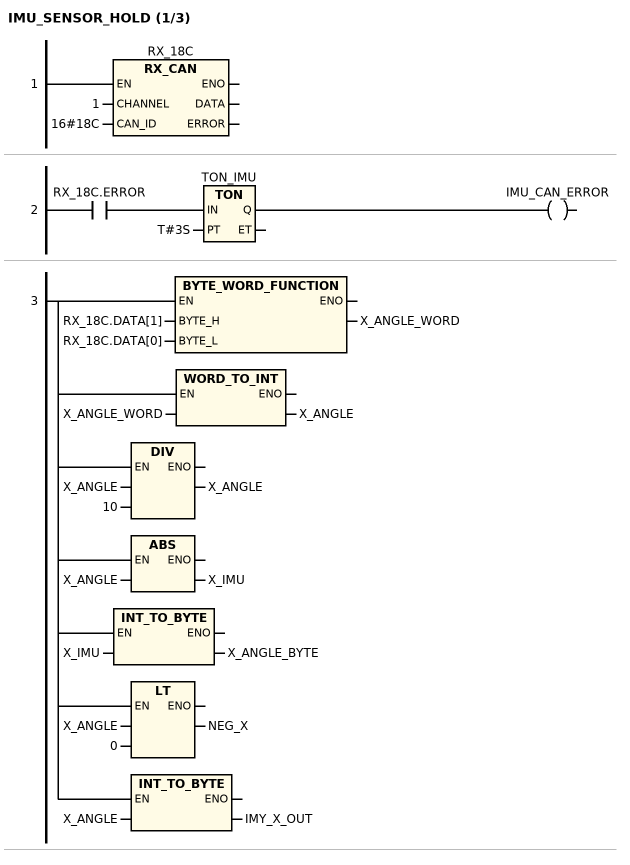
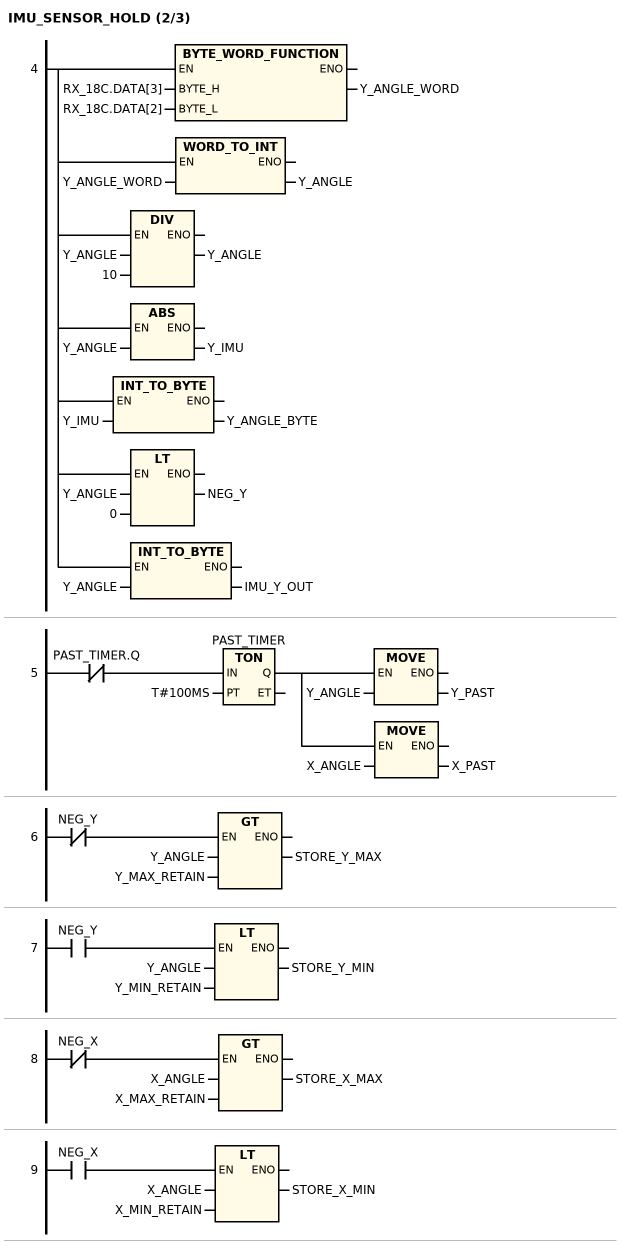
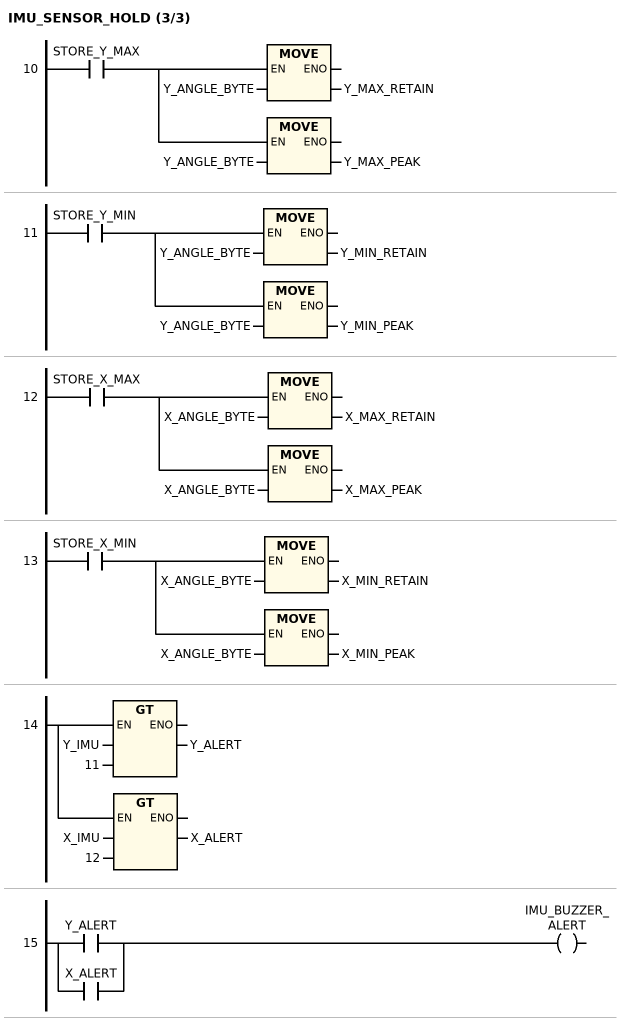
_LD_ (* Ladder Diagram *)
NETWORK 1
	*
		EN --- RX_18C:RX_CAN(CHANNEL: 1, CAN_ID: 16#18C)
NETWORK 2
	[RX_18C.ERROR] - TON_IMU:TON(IN: *, PT: T#3S) --- (IMU_CAN_ERROR)
NETWORK 3
	*
		EN --- BYTE_WORD_FUNCTION(BYTE_H: RX_18C.DATA[1], BYTE_L: RX_18C.DATA[0]) => X_ANGLE_WORD
		EN --- WORD_TO_INT(X_ANGLE_WORD) => X_ANGLE
		EN --- DIV(X_ANGLE, 10) => X_ANGLE
		EN --- ABS(X_ANGLE) => X_IMU
		EN --- INT_TO_BYTE(X_IMU) => X_ANGLE_BYTE
		EN --- LT(X_ANGLE, 0) => NEG_X
		EN --- INT_TO_BYTE(X_ANGLE) => IMY_X_OUT
NETWORK 4
	*
		EN --- BYTE_WORD_FUNCTION(BYTE_H: RX_18C.DATA[3], BYTE_L: RX_18C.DATA[2]) => Y_ANGLE_WORD
		EN --- WORD_TO_INT(Y_ANGLE_WORD) => Y_ANGLE
		EN --- DIV(Y_ANGLE, 10) => Y_ANGLE
		EN --- ABS(Y_ANGLE) => Y_IMU
		EN --- INT_TO_BYTE(Y_IMU) => Y_ANGLE_BYTE
		EN --- LT(Y_ANGLE, 0) => NEG_Y
		EN --- INT_TO_BYTE(Y_ANGLE) => IMU_Y_OUT
NETWORK 5
	[/PAST_TIMER.Q] - PAST_TIMER:TON(IN: *, PT: T#100MS)
		EN --- MOVE(Y_ANGLE) => Y_PAST
		EN --- MOVE(X_ANGLE) => X_PAST
NETWORK 6
	[/NEG_Y]
		EN --- GT(Y_ANGLE, Y_MAX_RETAIN) => STORE_Y_MAX
NETWORK 7
	[NEG_Y]
		EN --- LT(Y_ANGLE, Y_MIN_RETAIN) => STORE_Y_MIN
NETWORK 8
	[/NEG_X]
		EN --- GT(X_ANGLE, X_MAX_RETAIN) => STORE_X_MAX
NETWORK 9
	[NEG_X]
		EN --- LT(X_ANGLE, X_MIN_RETAIN) => STORE_X_MIN
NETWORK 10
	[STORE_Y_MAX]
		EN --- MOVE(Y_ANGLE_BYTE) => Y_MAX_RETAIN
		EN --- MOVE(Y_ANGLE_BYTE) => Y_MAX_PEAK
NETWORK 11
	[STORE_Y_MIN]
		EN --- MOVE(Y_ANGLE_BYTE) => Y_MIN_RETAIN
		EN --- MOVE(Y_ANGLE_BYTE) => Y_MIN_PEAK
NETWORK 12
	[STORE_X_MAX]
		EN --- MOVE(X_ANGLE_BYTE) => X_MAX_RETAIN
		EN --- MOVE(X_ANGLE_BYTE) => X_MAX_PEAK
NETWORK 13
	[STORE_X_MIN]
		EN --- MOVE(X_ANGLE_BYTE) => X_MIN_RETAIN
		EN --- MOVE(X_ANGLE_BYTE) => X_MIN_PEAK
NETWORK 14
	*
		EN --- GT(Y_IMU, 11) => Y_ALERT
		EN --- GT(X_IMU, 12) => X_ALERT
NETWORK 15
	{ [Y_ALERT] | [X_ALERT] } --- (IMU_BUZZER_ALERT)
_END_LD_
(* the same logic as Structured Text *)
(* Network 1 *)
RX_18C(CHANNEL := 1, CAN_ID := 16#18C);
(* Network 2 *)
TON_IMU(IN := RX_18C.ERROR, PT := T#3S);
IMU_CAN_ERROR := TON_IMU.Q;
(* Network 3 *)
X_ANGLE_WORD := BYTE_WORD_FUNCTION(BYTE_H := RX_18C.DATA[1], BYTE_L := RX_18C.DATA[0]);
X_ANGLE := WORD_TO_INT(X_ANGLE_WORD);
X_ANGLE := X_ANGLE / 10;
X_IMU := ABS(X_ANGLE);
X_ANGLE_BYTE := INT_TO_BYTE(X_IMU);
NEG_X := X_ANGLE < 0;
IMY_X_OUT := INT_TO_BYTE(X_ANGLE);
(* Network 4 *)
Y_ANGLE_WORD := BYTE_WORD_FUNCTION(BYTE_H := RX_18C.DATA[3], BYTE_L := RX_18C.DATA[2]);
Y_ANGLE := WORD_TO_INT(Y_ANGLE_WORD);
Y_ANGLE := Y_ANGLE / 10;
Y_IMU := ABS(Y_ANGLE);
Y_ANGLE_BYTE := INT_TO_BYTE(Y_IMU);
NEG_Y := Y_ANGLE < 0;
IMU_Y_OUT := INT_TO_BYTE(Y_ANGLE);
(* Network 5 *)
PAST_TIMER(IN := NOT PAST_TIMER.Q, PT := T#100MS);
IF PAST_TIMER.Q THEN
	Y_PAST := Y_ANGLE;
	X_PAST := X_ANGLE;
END_IF;
(* Network 6 *)
IF NOT NEG_Y THEN
	STORE_Y_MAX := Y_ANGLE > Y_MAX_RETAIN;
END_IF;
(* Network 7 *)
IF NEG_Y THEN
	STORE_Y_MIN := Y_ANGLE < Y_MIN_RETAIN;
END_IF;
(* Network 8 *)
IF NOT NEG_X THEN
	STORE_X_MAX := X_ANGLE > X_MAX_RETAIN;
END_IF;
(* Network 9 *)
IF NEG_X THEN
	STORE_X_MIN := X_ANGLE < X_MIN_RETAIN;
END_IF;
(* Network 10 *)
IF STORE_Y_MAX THEN
	Y_MAX_RETAIN := Y_ANGLE_BYTE;
	Y_MAX_PEAK := Y_ANGLE_BYTE;
END_IF;
(* Network 11 *)
IF STORE_Y_MIN THEN
	Y_MIN_RETAIN := Y_ANGLE_BYTE;
	Y_MIN_PEAK := Y_ANGLE_BYTE;
END_IF;
(* Network 12 *)
IF STORE_X_MAX THEN
	X_MAX_RETAIN := X_ANGLE_BYTE;
	X_MAX_PEAK := X_ANGLE_BYTE;
END_IF;
(* Network 13 *)
IF STORE_X_MIN THEN
	X_MIN_RETAIN := X_ANGLE_BYTE;
	X_MIN_PEAK := X_ANGLE_BYTE;
END_IF;
(* Network 14 *)
Y_ALERT := Y_IMU > 11;
X_ALERT := X_IMU > 12;
(* Network 15 *)
IMU_BUZZER_ALERT := Y_ALERT OR X_ALERT;
END_FUNCTION_BLOCK

(* POU PROGRAM_FBs/MAKERSAN_JOYSTICK, LD *)
FUNCTION_BLOCK MAKERSAN_JOYSTICK
(*
Created by: SR Karthik Raju
Date: 23-09-24
Version: 1
Updated by:
Update date:
Description: This block reads the Makersan joystick data from the CAN.
*)
VAR_INPUT
	CAN_CHANNEL: BYTE;
END_VAR
VAR_OUTPUT
	JX: INT;
	JY: INT;
	LEFT_BUTTON: BOOL;
	RIGHT_BUTTON: BOOL;
	DEADMAN: BOOL;
	AXIS_POSITION: ARRAY [0..4] OF BOOL;
	CAN_ERROR: BOOL;
END_VAR
VAR
	RX_284: RX_CAN;
	RX_184: RX_CAN;
	TON_1: TON;
	X_WORD: WORD;
	Y_WORD: WORD;
	JX_INT: INT;
	JY_INT: INT;
	JY_ORIGIN: BOOL;
	JX_ORIGIN: BOOL;
END_VAR
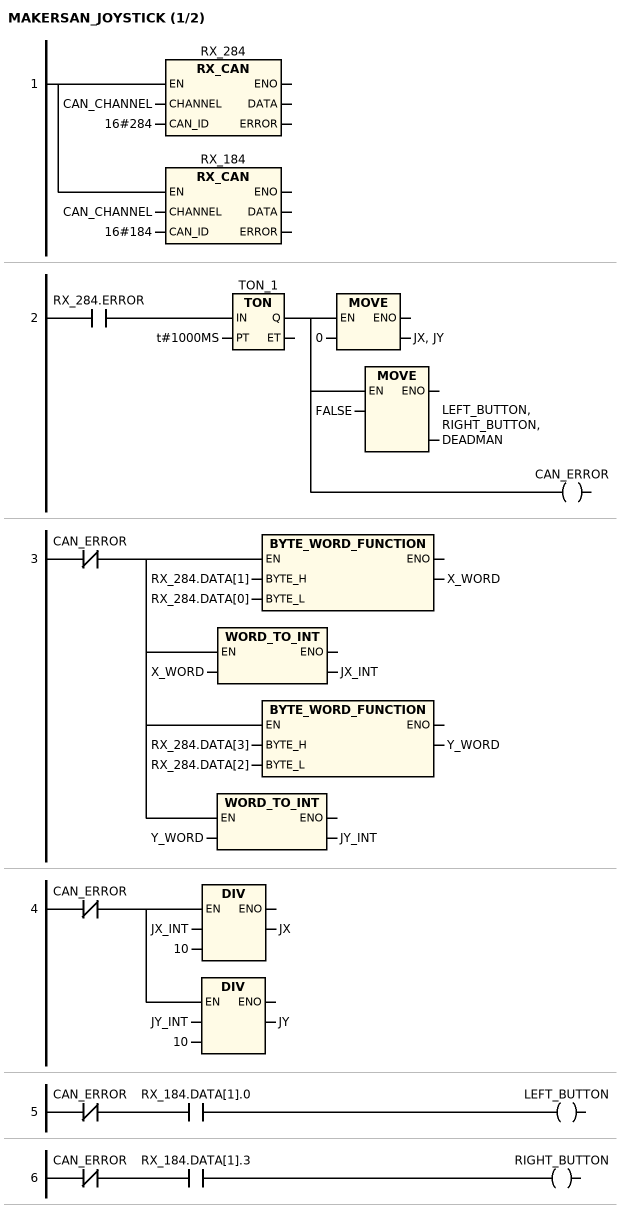
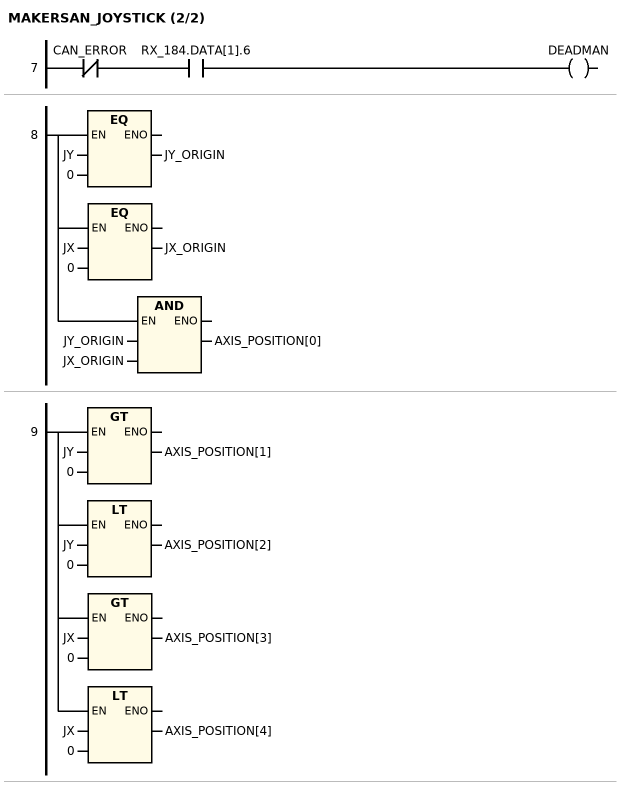
_LD_ (* Ladder Diagram *)
NETWORK 1
	*
		EN --- RX_284:RX_CAN(CHANNEL: CAN_CHANNEL, CAN_ID: 16#284)
		EN --- RX_184:RX_CAN(CHANNEL: CAN_CHANNEL, CAN_ID: 16#184)
NETWORK 2
	[RX_284.ERROR] - TON_1:TON(IN: *, PT: t#1000MS) --- (CAN_ERROR)
		EN --- MOVE(0) => JX, JY
		EN --- MOVE(FALSE) => LEFT_BUTTON, RIGHT_BUTTON, DEADMAN
NETWORK 3
	[/CAN_ERROR]
		EN --- BYTE_WORD_FUNCTION(BYTE_H: RX_284.DATA[1], BYTE_L: RX_284.DATA[0]) => X_WORD
		EN --- WORD_TO_INT(X_WORD) => JX_INT
		EN --- BYTE_WORD_FUNCTION(BYTE_H: RX_284.DATA[3], BYTE_L: RX_284.DATA[2]) => Y_WORD
		EN --- WORD_TO_INT(Y_WORD) => JY_INT
NETWORK 4
	[/CAN_ERROR]
		EN --- DIV(JX_INT, 10) => JX
		EN --- DIV(JY_INT, 10) => JY
NETWORK 5
	[/CAN_ERROR] - [RX_184.DATA[1].0] --- (LEFT_BUTTON)
NETWORK 6
	[/CAN_ERROR] - [RX_184.DATA[1].3] --- (RIGHT_BUTTON)
NETWORK 7
	[/CAN_ERROR] - [RX_184.DATA[1].6] --- (DEADMAN)
NETWORK 8
	*
		EN --- EQ(JY, 0) => JY_ORIGIN
		EN --- EQ(JX, 0) => JX_ORIGIN
		EN --- AND(JY_ORIGIN, JX_ORIGIN) => AXIS_POSITION[0]
NETWORK 9
	*
		EN --- GT(JY, 0) => AXIS_POSITION[1]
		EN --- LT(JY, 0) => AXIS_POSITION[2]
		EN --- GT(JX, 0) => AXIS_POSITION[3]
		EN --- LT(JX, 0) => AXIS_POSITION[4]
_END_LD_
(* the same logic as Structured Text *)
(* Network 1 *)
RX_284(CHANNEL := CAN_CHANNEL, CAN_ID := 16#284);
RX_184(CHANNEL := CAN_CHANNEL, CAN_ID := 16#184);
(* Network 2: see the listing above *)
(* Network 3 *)
IF NOT CAN_ERROR THEN
	X_WORD := BYTE_WORD_FUNCTION(BYTE_H := RX_284.DATA[1], BYTE_L := RX_284.DATA[0]);
	JX_INT := WORD_TO_INT(X_WORD);
	Y_WORD := BYTE_WORD_FUNCTION(BYTE_H := RX_284.DATA[3], BYTE_L := RX_284.DATA[2]);
	JY_INT := WORD_TO_INT(Y_WORD);
END_IF;
(* Network 4 *)
IF NOT CAN_ERROR THEN
	JX := JX_INT / 10;
	JY := JY_INT / 10;
END_IF;
(* Network 5 *)
LEFT_BUTTON := NOT CAN_ERROR AND RX_184.DATA[1].0;
(* Network 6 *)
RIGHT_BUTTON := NOT CAN_ERROR AND RX_184.DATA[1].3;
(* Network 7 *)
DEADMAN := NOT CAN_ERROR AND RX_184.DATA[1].6;
(* Network 8 *)
JY_ORIGIN := JY = 0;
JX_ORIGIN := JX = 0;
AXIS_POSITION[0] := JY_ORIGIN AND JX_ORIGIN;
(* Network 9 *)
AXIS_POSITION[1] := JY > 0;
AXIS_POSITION[2] := JY < 0;
AXIS_POSITION[3] := JX > 0;
AXIS_POSITION[4] := JX < 0;
END_FUNCTION_BLOCK

(* POU FUNCTIONS/MAP_INT, ST *)
FUNCTION MAP_INT : INT
(*
Created By: Nikshitha S
Date: 10-08-2023
Version: 1
Description: This function block maps the Input value range to the Output value range for the values in INT datatype.
Thus, consuming less memory than the library block "LIN_TRAFO" which uses REAL datatype.
*)
VAR_INPUT
	IN: INT;
	IN_MIN:INT;
	IN_MAX : INT;
	OUT_MIN:INT;
	OUT_MAX:INT;
END_VAR
VAR
	ERROR: BOOL;
	FINAL_MAP: INT;
	INPUT_RANGE: INT;
	OUTPUT_RANGE: INT;
END_VAR
ERROR := (IN_MAX-IN_MIN=0) OR (IN<IN_MIN) OR (IN>IN_MAX);
INPUT_RANGE := IN_MAX-IN_MIN;
OUTPUT_RANGE := OUT_MAX-OUT_MIN;
MAP_INT:= ((IN-IN_MIN)*OUTPUT_RANGE) / INPUT_RANGE + OUT_MIN;
IF ERROR AND (IN<IN_MIN)THEN
MAP_INT:=OUT_MIN;
END_IF
IF ERROR AND (IN>IN_MAX)THEN
MAP_INT:=OUT_MAX;
END_IF
END_FUNCTION

(* POU EXCLUDES/MAP_REAL, ST *)
FUNCTION MAP_REAL : REAL
(*
Created By: Bhagyesh
Date: Nov - 2021
Description: This function block maps the Input value range to the Output value range for the values in REAL datatype.
*)
VAR_INPUT
	IN: REAL;				(* input value*)
	IN_MIN:REAL;			(* minimum input value *)
	IN_MAX:REAL;			(* maximum input value *)
	OUT_MIN:REAL;		(* corresponding minimum output value *)
	OUT_MAX:REAL;		(* corresponding maximum output value *)
END_VAR
VAR
	Diff: REAL;
	ERROR: BOOL;		(* error: IN_MIN = IN_MAX or IN out of interval *)
END_VAR
Diff := IN_MAX-IN_MIN;
ERROR := (Diff=0) OR (IN<IN_MIN) OR (IN>IN_MAX);
MAP_REAL:= (IN-IN_MIN)/Diff * (OUT_MAX-OUT_MIN) + OUT_MIN;
IF ERROR AND (IN<IN_MIN)THEN
MAP_REAL:=OUT_MIN;
END_IF
IF ERROR AND (IN>IN_MAX)THEN
MAP_REAL:=OUT_MAX;
END_IF
END_FUNCTION

(* POU PROGRAM_FBs/THROTTLE_LOGIC, LD *)
FUNCTION_BLOCK THROTTLE_LOGIC
(*
Author: Bhagyesh
Description: This function block takes the joystick input from the RunLogic block and calculates the throttle for each side of the motors based on the turning logic.
This function block also implements the Zero degree turn.
*)
VAR_INPUT
	JX_IN: INT;
	JY_IN: INT;
	MCUBRAKE: BOOL;
	RPM_FACTOR_IN: INT;
END_VAR
VAR_OUTPUT
	THR_L: INT;
	THR_R: INT;
END_VAR
VAR
	THR_1: INT;
	THR_2: INT;
	THR_R_INTER: INT;
	SET_FWD: BOOL;
	SET_REV: BOOL;
	SET_RIGHT_ZERO: BOOL;
	SET_LEFT_ZERO: BOOL;

	JOY_ORIGIN: BOOL;
	FWD: BOOL;
	REV: BOOL;
	RIGHT_ZERO: BOOL;
	LEFT_ZERO: BOOL;
END_VAR
VAR CONSTANT

END_VAR
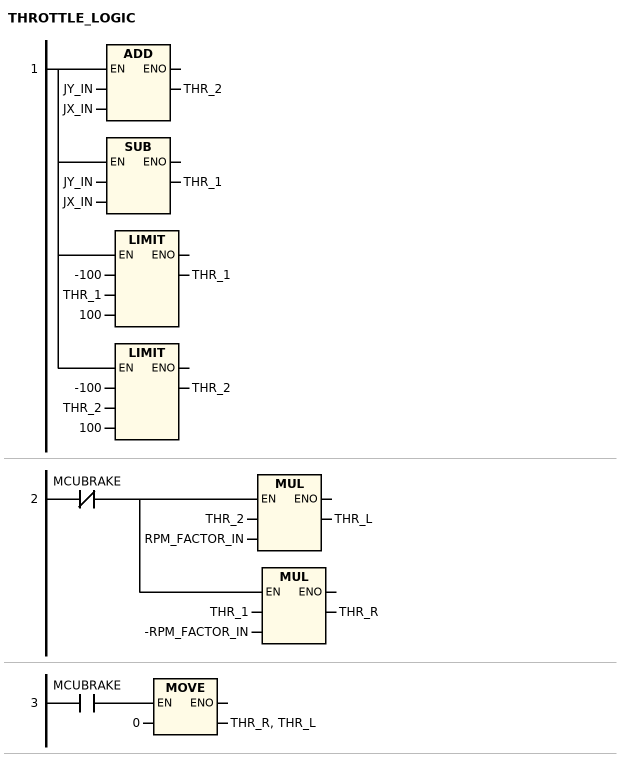
_LD_ (* Ladder Diagram *)
NETWORK 1
	*
		EN --- ADD(JY_IN, JX_IN) => THR_2
		EN --- SUB(JY_IN, JX_IN) => THR_1
		EN --- LIMIT(-100, THR_1, 100) => THR_1
		EN --- LIMIT(-100, THR_2, 100) => THR_2
NETWORK 2
	[/MCUBRAKE]
		EN --- MUL(THR_2, RPM_FACTOR_IN) => THR_L
		EN --- MUL(THR_1, -RPM_FACTOR_IN) => THR_R
NETWORK 3
	[MCUBRAKE]
		EN --- MOVE(0) => THR_R, THR_L
_END_LD_
(* the same logic as Structured Text *)
(* Network 1 *)
THR_2 := JY_IN + JX_IN;
THR_1 := JY_IN - JX_IN;
THR_1 := LIMIT(-100, THR_1, 100);
THR_2 := LIMIT(-100, THR_2, 100);
(* Network 2 *)
IF NOT MCUBRAKE THEN
	THR_L := THR_2 * RPM_FACTOR_IN;
	THR_R := THR_1 * (-RPM_FACTOR_IN);
END_IF;
(* Network 3: see the listing above *)
END_FUNCTION_BLOCK

(* Visualisation GLX_v3
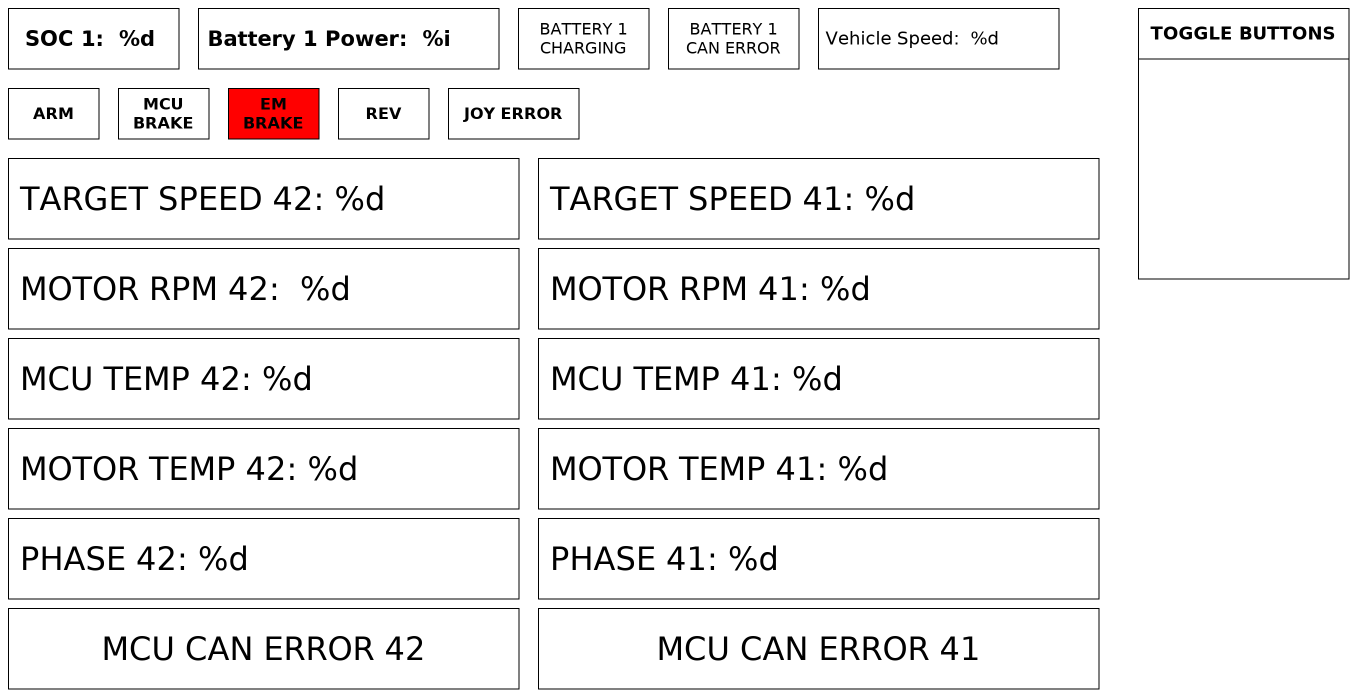
rounded rectangle at (10,10)-(181,71): text "SOC 1:  %d"; shows .BATTERY1_SOC
rounded rectangle at (200,10)-(501,71): text "Battery 1 Power:  %i"; shows .BATTERY1_POWER
rounded rectangle at (820,10)-(1061,71): text "Vehicle Speed:  %d"; shows .SPEED
rounded rectangle at (10,90)-(101,141): text "ARM"; alarm colour if .MCU_IGNITION
rounded rectangle at (120,90)-(211,141): text "MCU / BRAKE"; alarm colour if .MCU_BRAKE
rounded rectangle at (230,90)-(321,141): text "EM / BRAKE"; alarm colour if .EM_BRAKE
rounded rectangle at (540,250)-(1101,331): text "MOTOR RPM 41: %d"; shows .MOTOR_RPM[1]
rounded rectangle at (10,250)-(521,331): text "MOTOR RPM 42:  %d"; shows .MOTOR_RPM[2]
rounded rectangle at (540,340)-(1101,421): text "MCU TEMP 41: %d"; shows .MCU_TEMPERATURE[1]
rounded rectangle at (10,340)-(521,421): text "MCU TEMP 42: %d"; shows .MCU_TEMPERATURE[2]
rounded rectangle at (540,520)-(1101,601): text "PHASE 41: %d"; shows .MOTOR_PHASE_CURRENT[1]
rounded rectangle at (10,520)-(521,601): text "PHASE 42: %d"; shows .MOTOR_PHASE_CURRENT[2]
rounded rectangle at (540,160)-(1101,241): text "TARGET SPEED 41: %d"; shows .MOTOR_TARGET_RPM[1]
rounded rectangle at (10,160)-(521,241): text "TARGET SPEED 42: %d"; shows .MOTOR_TARGET_RPM[2]
rounded rectangle at (450,90)-(581,141): text "JOY ERROR"; alarm colour if .JOY_ERROR
rounded rectangle at (10,610)-(521,691): text "MCU CAN ERROR 42"; alarm colour if .MCU_CAN_ERROR[2]
rounded rectangle at (670,10)-(801,71): text "BATTERY 1 / CAN ERROR"; alarm colour if .BATTERY1_CAN_ERROR
rounded rectangle at (340,90)-(431,141): text "REV"; alarm colour if .REVERSE
rounded rectangle at (520,10)-(651,71): text "BATTERY 1 / CHARGING"; alarm colour if .BATTERY1_CHARGING
rounded rectangle at (540,610)-(1101,691): text "MCU CAN ERROR 41"; alarm colour if .MCU_CAN_ERROR[1]
rounded rectangle at (540,430)-(1101,511): text "MOTOR TEMP 41: %d"; shows .MOTOR_TEMPERATURE[1]
rounded rectangle at (10,430)-(521,511): text "MOTOR TEMP 42: %d"; shows .MOTOR_TEMPERATURE[2]
rectangle at (1140,10)-(1351,61): text "TOGGLE BUTTONS"
1 more shapes without text or variables
*)
